FUNCTION_BLOCK IDeviceEncode (* Composite Function Block Type *)
  (* Standard: 61499-2 *)
  (* Version 0.0, 6/12/2026, Schneider Electric, template *)
  PACKAGE SE.Nereda;
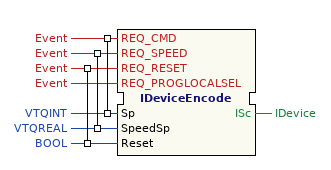
  EVENT_INPUT
    REQ_CMD WITH Sp; (* Request for new command *)
    REQ_SPEED WITH SpeedSp; (* Request for new  analog setpoint *)
    REQ_RESET WITH Reset; (* Request to reset the device *)
    REQ_PROGLOCALSEL; (* Request for program local owner *)
  END_EVENT
  VAR_INPUT
    Sp : VTQINT; (* Device setpoint in program local owner *)
    SpeedSp : VTQREAL; (* Device setpoint 1 in program local owner( in real) *)
    Reset : BOOL; (* 1= Reset command *)
  END_VAR
  PLUGS
    ISc : IDevice(ProgLocalSel := TRUE);
  END_PLUGS
  FBS
    CMD : RetriggerEvent(pin_CFF51EFF0A91DC53 := 3, pin_FDD5DC24A8674AF6 := T#1s);
    CMD_Merge : E_MERGE;
  END_FBS
  EVENT_CONNECTIONS
    REQ_SPEED TO ISc.REQ_SP;
    REQ_RESET TO ISc.REQ_RESET;
    REQ_PROGLOCALSEL TO ISc.REQ_PROGLOCALSEL;
    REQ_CMD TO CMD.2BC1963D96179493;
    CMD_Merge.EO TO ISc.REQ_CMD;
    CMD.4002AEF0814D09CF TO CMD_Merge.EI1;
    REQ_CMD TO CMD_Merge.EI2;
    ISc.CNF_READY TO CMD.2BC1963D96179493;
  END_CONNECTIONS
  DATA_CONNECTIONS
    Sp TO ISc.Lsp;
    SpeedSp TO ISc.LspReal1;
    Reset TO ISc.Reset;
  END_CONNECTIONS
END_FUNCTION_BLOCK
